{attribute addProperty BoxType "EP2339-0021-0019"}
{attribute addProperty Id "ChannelAT %I*ARRAY[0..15] OF Channel_E4AEF59E128160Channel_1AT %Q*ARRAY[0..15] OF Channel_7F374EB0128160WcStateAT %I*WcState_98A4DF7520.250InfoDataAT %I*InfoData_192954DE1620"}
{attribute addProperty CRC "4216243017"}
{attribute addProperty SizeInBites "274"}
{attribute addProperty SizeInBytes "34.25"}
TYPE EP2339_9219B498 :
STRUCT
	{attribute addProperty Name "Channel"}
	Channel : ARRAY[0..15] OF Channel_E4AEF59E;
	{attribute addProperty Name "Channel_1"}
	Channel_1 : ARRAY[0..15] OF Channel_7F374EB0;
	{attribute addProperty Name "WcState"}
	WcState : WcState_98A4DF75;
	{attribute addProperty Name "InfoData"}
	InfoData : InfoData_192954DE;
END_STRUCT
END_TYPE

(* stored: Version 1.2.0.0, ProductVersion 3.1.4024.9
   DUT EP2339_9219B498: Id {b30dee69-1358-429f-9aba-d0e5b2b064e0} *)
